FUNCTION_BLOCK CiA_DS402Statusword_Vacon EXTENDS CiA_DS402Statusword
VAR_INPUT
END_VAR
VAR_OUTPUT	
	TargetReached				: BOOL; // Bit 10 commonly used FOR in target position, velocity ect.
	IncorrectDriveMode		:	BOOL; //Manufacturer specific_Bit14
END_VAR

METHOD PUBLIC readStatusword : BOOL
VAR_INPUT
	Statusword 					:	UINT;
END_VAR


	TargetReached											:= Statusword.10;

	IncorrectDriveMode										:= Statusword.14;


	readStatusword											:= SUPER^.readStatusword(Statusword);
END_METHOD

END_FUNCTION_BLOCK

(* stored: Version 1.1.0.1, ProductVersion 3.1.4024.3
   POU CiA_DS402Statusword_Vacon: Id {c225f227-090c-464a-94f1-32ccef406c32}, SpecialFunc None
   Method readStatusword: Id {64fca09e-e8e7-4463-b099-62aa5eacfe60} *)
